GLOBALCONSTANTS IG1_Device_Classes (* Industry Group 1 specific device classes (vehicle systems) *)
  (* Standard: 61499-1 *)
  (* Version 1.0, 2026-06-30, Franz Höpfinger, Demmler Andreas Fahrzeugbau *)
  PACKAGE isobus::pgn::const;
  VAR_GLOBAL CONSTANT
    DC_NON_SPECIFIC_SYSTEM : BYTE := 0; (* Device Class / Vehicle System: Non-specific System *)
    DC_TRACTOR : BYTE := 1; (* Device Class / Vehicle System: Tractor *)
    DC_TRAILER : BYTE := 2; (* Device Class / Vehicle System: Trailer *)
    DC_NOT_AVAILABLE : BYTE := 127; (* Device Class / Vehicle System: Not Available *)
  END_VAR
END_GLOBALCONSTANTS
